FUNCTION_BLOCK AI_16 (* Composite Function Block Type *)
  (* Standard: 61499-2 *)
  (* Version 0.0, 2018-12-21, 4DIAC-IDE, 4DIAC-Consortium *)
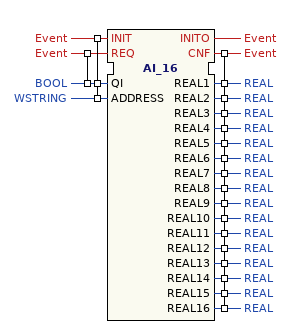
  EVENT_INPUT
    INIT WITH QI, ADDRESS; (* Initialization Request *)
    REQ WITH QI; (* Normal Execution Request *)
  END_EVENT
  EVENT_OUTPUT
    INITO; (* Initialization Confirm *)
    CNF WITH REAL1, REAL2, REAL3, REAL4, REAL5, REAL6, REAL7, REAL8, REAL9, REAL10, REAL11, REAL12, REAL13, REAL14, REAL15, REAL16; (* Execution Confirmation *)
  END_EVENT
  VAR_INPUT
    QI : BOOL;
    ADDRESS : WSTRING;
  END_VAR
  VAR_OUTPUT
    REAL1 : REAL;
    REAL2 : REAL;
    REAL3 : REAL;
    REAL4 : REAL;
    REAL5 : REAL;
    REAL6 : REAL;
    REAL7 : REAL;
    REAL8 : REAL;
    REAL9 : REAL;
    REAL10 : REAL;
    REAL11 : REAL;
    REAL12 : REAL;
    REAL13 : REAL;
    REAL14 : REAL;
    REAL15 : REAL;
    REAL16 : REAL;
  END_VAR
  FBS
    AdressInputAnalog1 : F_CONCAT;
    InputAnalog1 : SUBSCRIBE_1;
    InputAnalog3 : SUBSCRIBE_1;
    InputAnalog2 : SUBSCRIBE_1;
    InputAnalog4 : SUBSCRIBE_1;
    InputAnalog5 : SUBSCRIBE_1;
    AdressInputAnalog2 : F_CONCAT;
    AdressInputAnalog3 : F_CONCAT;
    AdressInputAnalog4 : F_CONCAT;
    AdressInputAnalog6 : F_CONCAT;
    AdressInputAnalog7 : F_CONCAT;
    AdressInputAnalog8 : F_CONCAT;
    AdressInputAnalog9 : F_CONCAT;
    AdressInputAnalog10 : F_CONCAT;
    AdressInputAnalog11 : F_CONCAT;
    AdressInputAnalog12 : F_CONCAT;
    AdressInputAnalog13 : F_CONCAT;
    AdressInputAnalog14 : F_CONCAT;
    AdressInputAnalog15 : F_CONCAT;
    AdressInputAnalog16 : F_CONCAT;
    AdressInputAnalog5 : F_CONCAT;
    PortInputAnalog1 : WSTRING2WSTRING(IN := :61000);
    PortInputAnalog2 : WSTRING2WSTRING(IN := :61001);
    PortInputAnalog4 : WSTRING2WSTRING(IN := :61003);
    PortInputAnalog3 : WSTRING2WSTRING(IN := :61002);
    PortInputAnalog5 : WSTRING2WSTRING(IN := :61004);
    PortInputAnalog6 : WSTRING2WSTRING(IN := :61005);
    PortInputAnalog7 : WSTRING2WSTRING(IN := :61006);
    PortInputAnalog8 : WSTRING2WSTRING(IN := :61007);
    PortInputAnalog9 : WSTRING2WSTRING(IN := :61008);
    PortInputAnalog10 : WSTRING2WSTRING(IN := :61009);
    PortInputAnalog11 : WSTRING2WSTRING(IN := :61010);
    PortInputAnalog12 : WSTRING2WSTRING(IN := :61011);
    PortInputAnalog13 : WSTRING2WSTRING(IN := :61012);
    PortInputAnalog14 : WSTRING2WSTRING(IN := :61013);
    PortInputAnalog15 : WSTRING2WSTRING(IN := :61014);
    WSTRING2WSTRING_15 : WSTRING2WSTRING(IN := :61015);
    InputAnalog6 : SUBSCRIBE_1;
    InputAnalog7 : SUBSCRIBE_1;
    InputAnalog8 : SUBSCRIBE_1;
    InputAnalog9 : SUBSCRIBE_1;
    InputAnalog10 : SUBSCRIBE_1;
    InputAnalog11 : SUBSCRIBE_1;
    InputAnalog12 : SUBSCRIBE_1;
    InputAnalog13 : SUBSCRIBE_1;
    InputAnalog14 : SUBSCRIBE_1;
    InputAnalog15 : SUBSCRIBE_1;
    InitoInput16 : E_Merge16;
    CNFInput16 : E_Merge16;
    InputAnalog16 : SUBSCRIBE_1;
  END_FBS
  EVENT_CONNECTIONS
    AdressInputAnalog1.CNF TO InputAnalog1.RSP;
    AdressInputAnalog2.CNF TO InputAnalog2.RSP;
    AdressInputAnalog3.CNF TO InputAnalog3.RSP;
    AdressInputAnalog4.CNF TO InputAnalog4.RSP;
    AdressInputAnalog5.CNF TO InputAnalog5.RSP;
    INIT TO InputAnalog1.INIT;
    INIT TO InputAnalog2.INIT;
    INIT TO InputAnalog3.INIT;
    INIT TO InputAnalog4.INIT;
    INIT TO InputAnalog5.INIT;
    PortInputAnalog1.CNF TO AdressInputAnalog1.REQ;
    INIT TO PortInputAnalog1.REQ;
    PortInputAnalog2.CNF TO AdressInputAnalog2.REQ;
    INIT TO PortInputAnalog2.REQ;
    INIT TO PortInputAnalog3.REQ;
    PortInputAnalog3.CNF TO AdressInputAnalog3.REQ;
    INIT TO PortInputAnalog4.REQ;
    INIT TO AdressInputAnalog4.REQ;
    INIT TO PortInputAnalog5.REQ;
    PortInputAnalog5.CNF TO AdressInputAnalog5.REQ;
    INIT TO PortInputAnalog6.REQ;
    PortInputAnalog6.CNF TO AdressInputAnalog6.REQ;
    INIT TO PortInputAnalog7.REQ;
    PortInputAnalog7.CNF TO AdressInputAnalog7.REQ;
    INIT TO PortInputAnalog8.REQ;
    INIT TO PortInputAnalog9.REQ;
    PortInputAnalog9.CNF TO AdressInputAnalog9.REQ;
    INIT TO PortInputAnalog10.REQ;
    PortInputAnalog10.CNF TO AdressInputAnalog10.REQ;
    INIT TO PortInputAnalog11.REQ;
    PortInputAnalog11.CNF TO AdressInputAnalog11.REQ;
    INIT TO PortInputAnalog12.REQ;
    PortInputAnalog12.CNF TO AdressInputAnalog12.REQ;
    INIT TO PortInputAnalog13.REQ;
    PortInputAnalog13.CNF TO AdressInputAnalog13.REQ;
    INIT TO PortInputAnalog14.REQ;
    PortInputAnalog14.CNF TO AdressInputAnalog14.REQ;
    INIT TO WSTRING2WSTRING_15.REQ;
    INIT TO PortInputAnalog15.REQ;
    PortInputAnalog15.CNF TO AdressInputAnalog15.REQ;
    WSTRING2WSTRING_15.CNF TO AdressInputAnalog16.REQ;
    REQ TO InputAnalog1.RSP;
    REQ TO InputAnalog2.RSP;
    REQ TO InputAnalog3.RSP;
    REQ TO InputAnalog4.RSP;
    REQ TO InputAnalog5.RSP;
    INIT TO InputAnalog6.INIT;
    AdressInputAnalog6.CNF TO InputAnalog6.RSP;
    REQ TO InputAnalog6.RSP;
    AdressInputAnalog7.CNF TO InputAnalog7.RSP;
    PortInputAnalog8.CNF TO AdressInputAnalog8.REQ;
    AdressInputAnalog8.CNF TO InputAnalog8.RSP;
    AdressInputAnalog9.CNF TO InputAnalog9.RSP;
    AdressInputAnalog11.CNF TO InputAnalog11.RSP;
    AdressInputAnalog12.CNF TO InputAnalog12.RSP;
    AdressInputAnalog13.CNF TO InputAnalog13.RSP;
    AdressInputAnalog14.CNF TO InputAnalog14.RSP;
    AdressInputAnalog15.CNF TO InputAnalog15.RSP;
    INIT TO InputAnalog7.INIT;
    INIT TO InputAnalog8.INIT;
    INIT TO InputAnalog9.INIT;
    AdressInputAnalog10.CNF TO InputAnalog10.RSP;
    INIT TO InputAnalog10.INIT;
    INIT TO InputAnalog12.INIT;
    INIT TO InputAnalog11.INIT;
    INIT TO InputAnalog13.INIT;
    INIT TO InputAnalog14.INIT;
    INIT TO InputAnalog15.INIT;
    REQ TO InputAnalog7.RSP;
    REQ TO InputAnalog8.RSP;
    REQ TO InputAnalog9.RSP;
    REQ TO InputAnalog10.RSP;
    REQ TO InputAnalog11.RSP;
    REQ TO InputAnalog12.RSP;
    REQ TO InputAnalog13.RSP;
    REQ TO InputAnalog14.RSP;
    REQ TO InputAnalog15.RSP;
    InputAnalog1.INITO TO InitoInput16.EI1;
    InputAnalog2.INITO TO InitoInput16.EI2;
    InputAnalog3.INITO TO InitoInput16.EI3;
    InputAnalog4.INITO TO InitoInput16.EI4;
    InputAnalog5.INITO TO InitoInput16.EI5;
    InputAnalog6.INITO TO InitoInput16.EI6;
    InputAnalog7.INITO TO InitoInput16.EI7;
    InputAnalog8.INITO TO InitoInput16.EI8;
    InputAnalog9.INITO TO InitoInput16.EI9;
    InputAnalog10.INITO TO InitoInput16.EI10;
    InputAnalog11.INITO TO InitoInput16.EI11;
    InputAnalog12.INITO TO InitoInput16.EI12;
    InputAnalog13.INITO TO InitoInput16.EI13;
    InputAnalog14.INITO TO InitoInput16.EI14;
    InputAnalog15.INITO TO InitoInput16.EI15;
    InputAnalog1.IND TO CNFInput16.EI1;
    InputAnalog2.IND TO CNFInput16.EI2;
    InputAnalog3.IND TO CNFInput16.EI3;
    InputAnalog5.IND TO CNFInput16.EI5;
    InputAnalog6.IND TO CNFInput16.EI6;
    InputAnalog7.IND TO CNFInput16.EI7;
    InputAnalog8.IND TO CNFInput16.EI8;
    InputAnalog9.IND TO CNFInput16.EI9;
    InputAnalog10.IND TO CNFInput16.EI10;
    InputAnalog11.IND TO CNFInput16.EI11;
    InputAnalog12.IND TO CNFInput16.EI12;
    InputAnalog13.IND TO CNFInput16.EI13;
    InputAnalog14.IND TO CNFInput16.EI14;
    InputAnalog15.IND TO CNFInput16.EI15;
    InitoInput16.EO TO INITO;
    CNFInput16.EO TO CNF;
    AdressInputAnalog16.CNF TO InputAnalog16.RSP;
    INIT TO InputAnalog16.INIT;
    InputAnalog16.INITO TO InitoInput16.EI16;
    InputAnalog16.IND TO CNFInput16.EI16;
    InputAnalog4.IND TO CNFInput16.EI4;
  END_CONNECTIONS
  DATA_CONNECTIONS
    QI TO InputAnalog1.QI;
    QI TO InputAnalog3.QI;
    QI TO InputAnalog2.QI;
    QI TO InputAnalog4.QI;
    QI TO InputAnalog5.QI;
    AdressInputAnalog1.OUT TO InputAnalog1.ID;
    AdressInputAnalog2.OUT TO InputAnalog2.ID;
    AdressInputAnalog3.OUT TO InputAnalog3.ID;
    AdressInputAnalog4.OUT TO InputAnalog4.ID;
    AdressInputAnalog5.OUT TO InputAnalog5.ID;
    ADDRESS TO AdressInputAnalog1.IN1;
    ADDRESS TO AdressInputAnalog2.IN1;
    ADDRESS TO AdressInputAnalog3.IN1;
    ADDRESS TO AdressInputAnalog4.IN1;
    ADDRESS TO AdressInputAnalog5.IN1;
    ADDRESS TO AdressInputAnalog6.IN1;
    ADDRESS TO AdressInputAnalog7.IN1;
    ADDRESS TO AdressInputAnalog8.IN1;
    ADDRESS TO AdressInputAnalog9.IN1;
    ADDRESS TO AdressInputAnalog10.IN1;
    ADDRESS TO AdressInputAnalog11.IN1;
    ADDRESS TO AdressInputAnalog12.IN1;
    ADDRESS TO AdressInputAnalog15.IN1;
    ADDRESS TO AdressInputAnalog16.IN1;
    PortInputAnalog1.OUT TO AdressInputAnalog1.IN2;
    PortInputAnalog2.OUT TO AdressInputAnalog2.IN2;
    PortInputAnalog3.OUT TO AdressInputAnalog3.IN2;
    PortInputAnalog4.OUT TO AdressInputAnalog4.IN2;
    PortInputAnalog5.OUT TO AdressInputAnalog5.IN2;
    PortInputAnalog6.OUT TO AdressInputAnalog6.IN2;
    PortInputAnalog8.OUT TO AdressInputAnalog8.IN2;
    PortInputAnalog7.OUT TO AdressInputAnalog7.IN2;
    PortInputAnalog10.OUT TO AdressInputAnalog10.IN2;
    PortInputAnalog9.OUT TO AdressInputAnalog9.IN2;
    PortInputAnalog11.OUT TO AdressInputAnalog11.IN2;
    PortInputAnalog12.OUT TO AdressInputAnalog12.IN2;
    PortInputAnalog13.OUT TO AdressInputAnalog13.IN2;
    PortInputAnalog14.OUT TO AdressInputAnalog14.IN2;
    PortInputAnalog15.OUT TO AdressInputAnalog15.IN2;
    WSTRING2WSTRING_15.OUT TO AdressInputAnalog16.IN2;
    InputAnalog1.RD_1 TO REAL1;
    InputAnalog2.RD_1 TO REAL2;
    InputAnalog3.RD_1 TO REAL3;
    InputAnalog4.RD_1 TO REAL4;
    InputAnalog5.RD_1 TO REAL5;
    QI TO InputAnalog6.QI;
    AdressInputAnalog6.OUT TO InputAnalog6.ID;
    AdressInputAnalog7.OUT TO InputAnalog7.ID;
    AdressInputAnalog8.OUT TO InputAnalog8.ID;
    AdressInputAnalog9.OUT TO InputAnalog9.ID;
    AdressInputAnalog10.OUT TO InputAnalog10.ID;
    AdressInputAnalog11.OUT TO InputAnalog11.ID;
    AdressInputAnalog12.OUT TO InputAnalog12.ID;
    AdressInputAnalog13.OUT TO InputAnalog13.ID;
    AdressInputAnalog14.OUT TO InputAnalog14.ID;
    AdressInputAnalog15.OUT TO InputAnalog15.ID;
    ADDRESS TO AdressInputAnalog13.IN1;
    ADDRESS TO AdressInputAnalog14.IN1;
    QI TO InputAnalog7.QI;
    QI TO InputAnalog8.QI;
    QI TO InputAnalog9.QI;
    QI TO InputAnalog10.QI;
    QI TO InputAnalog11.QI;
    QI TO InputAnalog12.QI;
    QI TO InputAnalog13.QI;
    QI TO InputAnalog14.QI;
    QI TO InputAnalog15.QI;
    InputAnalog6.RD_1 TO REAL6;
    InputAnalog7.RD_1 TO REAL7;
    InputAnalog8.RD_1 TO REAL8;
    InputAnalog9.RD_1 TO REAL9;
    InputAnalog10.RD_1 TO REAL10;
    InputAnalog11.RD_1 TO REAL11;
    InputAnalog12.RD_1 TO REAL12;
    InputAnalog13.RD_1 TO REAL13;
    InputAnalog14.RD_1 TO REAL14;
    InputAnalog15.RD_1 TO REAL15;
    AdressInputAnalog16.OUT TO InputAnalog16.ID;
    QI TO InputAnalog16.QI;
    InputAnalog16.RD_1 TO REAL16;
  END_CONNECTIONS
END_FUNCTION_BLOCK
